ABB RAPID module: Wobj_wobj_JMora.mod

MODULE Wobj_wobj_JMora
	! Points are read in order of declaration.
  ! Please do not change the order of points!

  LOCAL PERS robtarget pWobj_O_PointX1:=[[229.874,-701.855,652.493],[0.271133,0.548542,0.754379,-0.237699],[-1,-1,0,0],[9E+9,9E+9,9E+9,9E+9,9E+9,9E+9]];
	LOCAL PERS robtarget pWobj_O_PointX2:=[[-78.7227,-713.458,644.242],[0.271131,0.548554,0.754372,-0.237695],[-2,0,-1,0],[9E+9,9E+9,9E+9,9E+9,9E+9,9E+9]];
	LOCAL PERS robtarget pWobj_O_PointY1:=[[228.824,-521.78,653.089],[0.271128,0.548561,0.754368,-0.237695],[-1,-1,0,0],[9E+9,9E+9,9E+9,9E+9,9E+9,9E+9]];
	TASK PERS wobjdata wobj_JMora:=[FALSE,TRUE,"",[[0,0,-20],[1,0,0,0]],[[235.598,-701.64,652.646],[0.0133311,-0.0188038,0.999733,0.0014809]]];

ENDMODULE
